// Converts a T_Size value to a INT value.
FUNCTION F_SizeToInt : INT // The converted INT value from the given T_Size.
VAR_INPUT
	Size : T_Size; // The input size to be converted.
END_VAR

F_SizeToDint := TO_INT(LIMIT(0, Size, TO_UDINT(GVL_TypeValueLimits.INT_MAX)));

END_FUNCTION

(* stored: Version 1.1.0.1
   POU F_SizeToInt: Id {f6a52b8f-1519-0aa6-3b0e-e1fb525bb0e8}, SpecialFunc None *)
